// TIA Portal V20 export
DATA_BLOCK "ControlNodes"   // DB144
// stored: MemoryReserve 100, Namespace Unit1.Em2
   VAR
      em : "LAF_typeEmControlNode";
      emstate { S7_SetPoint := 'True'} : "LUC_typeStates";
      cm : "Unit1.Em2.typeCmControlNode";
      citiMap1 : Struct
         PMC : "LER_PMC_Input_Data";
         FlexNet { S7_SetPoint := 'True'} : "LER_FlexNet_Data";
      END_STRUCT;
      citiMap2 : Struct
         PMC : "LER_PMC_Input_Data";
         FlexNet { S7_SetPoint := 'True'} : "LER_FlexNet_Data";
      END_STRUCT;
      jrOutPnPLeft : "Unit1.Em2.typeSequenceControlNode_jrOutPnPLeft";
      jrOutPnPRight : "Unit1.Em2.typeSequenceControlNode_jrOutPnPRight";
      emData { S7_SetPoint := 'True'} : "Unit1.Em2.typeEmDataControlNode";
      SpecialFunctionMode : Struct
         DryRun : Struct
            JRdetectPV : Array[0..15] of Bool;
         END_STRUCT;
      END_STRUCT;
      unitCommunication : "Unit1.Em2.typeUnitCommunicationControlNode";
      cmJROutPnPLeftSafetyPin : "LBC_typeDigitalSignalControlNode";
      cmJROutPnPLeftJRDetect : "LBC_typeDigitalSignalControlNode";
      cmJROutPnPRightSafetyPin : "LBC_typeDigitalSignalControlNode";
      cmJROutPnPRightJRDetect : "LBC_typeDigitalSignalControlNode";
      cmJROutPnPLeftAxisX : "LBC_typeAxis64PosControlNode";
      cmJROutPnPLeftAxisZ : "LBC_typeAxis64PosControlNode";
      cmJROutPnPRightAxisX : "LBC_typeAxis64PosControlNode";
      cmJROutPnPRightAxisZ : "LBC_typeAxis64PosControlNode";
      cmJROutPnPLeftClampOpenClose : "LBC_typeTwoWayActuatorControlNode";
      cmJROutPnPRightClampOpenClose : "LBC_typeTwoWayActuatorControlNode";
      cmPowerMeter : "LER_typePAC3220ControlNode";
   END_VAR
BEGIN
END_DATA_BLOCK
